FUNCTION_BLOCK earth_fault (* Basic Function Block Type *)
  (* Standard: 61499-2 *)
  (* Version 0.0, 3/23/2016, gulzha, nxtControl GmbH, Template *)
  (* Version 1.0, 22/02/2021, Badger, 4diac, Refactored and migrated to 4diac *)
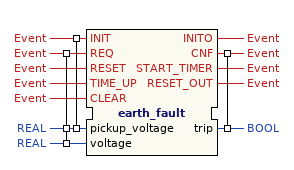
  EVENT_INPUT
    INIT WITH pickup_voltage; (* Initialization Request *)
    REQ WITH pickup_voltage, voltage; (* Normal Execution Request *)
    RESET;
    TIME_UP;
    CLEAR;
  END_EVENT
  EVENT_OUTPUT
    INITO; (* Initialisation confirmation *)
    CNF WITH trip; (* Execution Confirmation *)
    START_TIMER;
    RESET_OUT;
  END_EVENT
  VAR_INPUT
    pickup_voltage : REAL;
    voltage : REAL;
  END_VAR
  VAR_OUTPUT
    trip : BOOL;
  END_VAR
  VAR
    fault : BOOL; (* Ensures that the timer is started only once during a fault condition. *)
  END_VAR
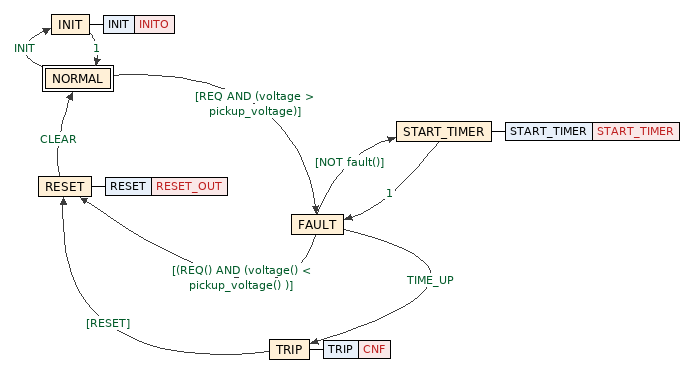
  EC_STATES
    NORMAL; (* Initial State *)
    INIT : INIT -> INITO; (* Initialization *)
    FAULT;
    TRIP : TRIP -> CNF;
    RESET : RESET -> RESET_OUT;
    START_TIMER : START_TIMER -> START_TIMER;
  END_STATES
  EC_TRANSITIONS
    NORMAL TO INIT := INIT;
    INIT TO NORMAL := 1;
    NORMAL TO FAULT := [REQ AND (voltage > pickup_voltage)];
    FAULT TO TRIP := TIME_UP;
    FAULT TO RESET := [(REQ() AND (voltage() < pickup_voltage() )]; (* Voltage has dropped back to a safe level so reset *)
    TRIP TO RESET := [RESET]; (* Clears the trip condition after the IED has been commanded to reset. *)
    FAULT TO START_TIMER := [NOT fault()]; (* If the timer has not already been started, then this is a new fault. Start the timer. *)
    START_TIMER TO FAULT := 1;
    RESET TO NORMAL := CLEAR;
  END_TRANSITIONS
  ALGORITHM INIT IN AnyText: (* Initialization algorithm *)
	trip() = false;
	fault() = false;
  END_ALGORITHM
  ALGORITHM REQ IN AnyText: (* Normally executed algorithm *)
	trip() = true;
  END_ALGORITHM
  ALGORITHM RESET IN AnyText:
;

trip := FALSE;
fault := FALSE;
  END_ALGORITHM
  ALGORITHM START_TIMER IN AnyText: (* Start timer after fault is detected *)
	fault() = true;
  END_ALGORITHM
  ALGORITHM TRIP IN AnyText: (* Trip after timeout. *)

  END_ALGORITHM
END_FUNCTION_BLOCK
